TYPE LoadCellI :
STRUCT
	AnalogSignal : INT;
	MaxSignalValue : INT;
	MaxUnitValue : INT;
END_STRUCT
END_TYPE

(* stored: Version 1.1.0.1, ProductVersion 3.1.4024.12
   DUT LoadCellI: Id {a0041e41-c42b-4712-b448-89813245e27d} *)
